Fanuc KAREL source: kc00044.KL

-- PROVISIONAL review KL for V1013-1; original PC SHA256 b4b27af20eab40e44e84bad982179195a94b4390d22a5e0f3cc7970a976e90ca
-- Incomplete behavior may be omitted. Consult companion uncertainty JSON. Do not deploy.
PROGRAM KC00044
%NOLOCKGROUP
BEGIN
  -- UNRESOLVED_PC offsets 5-39; opcodes 27,22,22,22,22,22,31
  -- UNRESOLVED_PC offsets 44-48; opcodes 7F
END KC00044
